{attribute addProperty BoxType "EL3162-0000-0019"}
{attribute addProperty Id "AI_Standard_ChannelAT %I*ARRAY[0..2] OF AI_Standard_Channel_087F71C76480WcStateAT %I*WcState_98A4DF7520.250InfoDataAT %I*InfoData_BC63D37F80100"}
{attribute addProperty CRC "3181681569"}
{attribute addProperty SizeInBites "146"}
{attribute addProperty SizeInBytes "18.25"}
TYPE EL3162_C6F348DD :
STRUCT
	{attribute addProperty Name "AI_Standard_Channel"}
	AI_Standard_Channel : ARRAY[0..2] OF AI_Standard_Channel_087F71C7;
	{attribute addProperty Name "WcState"}
	WcState : WcState_98A4DF75;
	{attribute addProperty Name "InfoData"}
	InfoData : InfoData_BC63D37F;
END_STRUCT
END_TYPE

(* stored: Version 1.2.0.0, ProductVersion 3.1.4024.9
   DUT EL3162_C6F348DD: Id {f2f62e93-54f0-40e2-b5c4-64107f70ad27} *)
